{region '#Template'}
	{attribute 'Version' := '6.0.0.0'}
	{attribute 'Tags' := '"LCID": "1031", "Text": "RA, Sunprotection, Sunblind, Zone"'}
	{attribute 'Tags' := '"LCID": "1033", "Text": "RA, Sunprotection, Sunblind, Zone"'}
	{attribute 'Using' := '"Type": "Template", "URI": "ST_BA_Facade"'}
	{attribute 'Using' := '"Type": "Template", "URI": "ST_BA_SunblindActuatorFeedback"'}
	{attribute 'Description' := '"LCID": "1031", "Text": "Sonnenschutzlogik (Jalousie) für eine Zone (Raum)"'}
	{attribute 'Description' := '"LCID": "1033", "Text": "Sunblind-logic (venetian blind) for one zone (room)"'}
{endregion}
FUNCTION_BLOCK FB_BA_SunblindZone EXTENDS FB_BA_Ext_SunblindAngle
VAR_INPUT	
	fRoomTempSen			: REAL;
	bPrcDetc				: BOOL;
	bSwiUp					: BOOL;
	bSwiDwn					: BOOL;	      
	stBuildingSpRmT			: ST_BA_SpRmT;
	stFacade				: ST_BA_Facade;
	stScene					: ST_BA_Sunbld;
	stReferenceFeedback		: ST_BA_SunblindActuatorFeedback;
END_VAR                 
VAR_OUTPUT              
	stSunBldOut				: ST_BA_SunBld;			// command telegram
END_VAR
VAR_INPUT CONSTANT PERSISTENT
	bThAutoSlcn				: BOOL;		// Thermo-automatic enable
	{attribute 'parameterUnit':= '%'}       
	fThAutoColPos			: REAL;		// Thermo-automatic cooling-position [%]
	{attribute 'parameterUnit':= 'degree'}  
	fThAutoColAngl			: REAL;		// Thermo-automatic cooling-angle [deg]
		                                    
	bSunPrtcSlcn			: BOOL;		// Sun-Protection-automatic enable     
		                                    
	bTwiLgtAutoSlcn			: BOOL;		// Twilight-automatic enable
	{attribute 'parameterUnit':= '%'}        
	fTwiLgtAutoPos			: REAL;		// Twilight-automatic cooling-position [%]
	{attribute 'parameterUnit':= 'degree'}   
	fTwiLgtAutoAngl			: REAL;		// Twilight-automatic cooling-angle [deg]
	{attribute 'parameterUnit':= 's'}
	{attribute 'parameterUnit':= 'ms'}
	nSwiOverTi 				: UDINT;	// zone-manual-control: switch-over time from step to continous mode [ms]
END_VAR
VAR_INPUT CONSTANT
	ManSwi					: FB_BA_SunBldSwi:= (ePrio:= E_BA_SunBldPrio.eManualGroup);
	ThAuto					: FB_BA_SunBldEvt:= (ePrio:= E_BA_SunBldPrio.eGroupThermoAuto);	
	SunPrtc					: FB_BA_SunBldEvt:= (ePrio:= E_BA_SunBldPrio.eSunProtection);	
	TwiLgtAuto				: FB_BA_SunBldEvt:= (ePrio:= E_BA_SunBldPrio.eGroupTwiLightAuto);
END_VAR
VAR                       	                                                    
	ThAutoSwi				: FB_BA_Swi2P;                                    
	PrioSwi					: FB_BA_SunBldTgmSel8;
	EnSunBldSwi				: SR;
END_VAR
VAR // added by the converter: edge detectors and wires of the graphical bodies
    _w1 : BOOL;
END_VAR

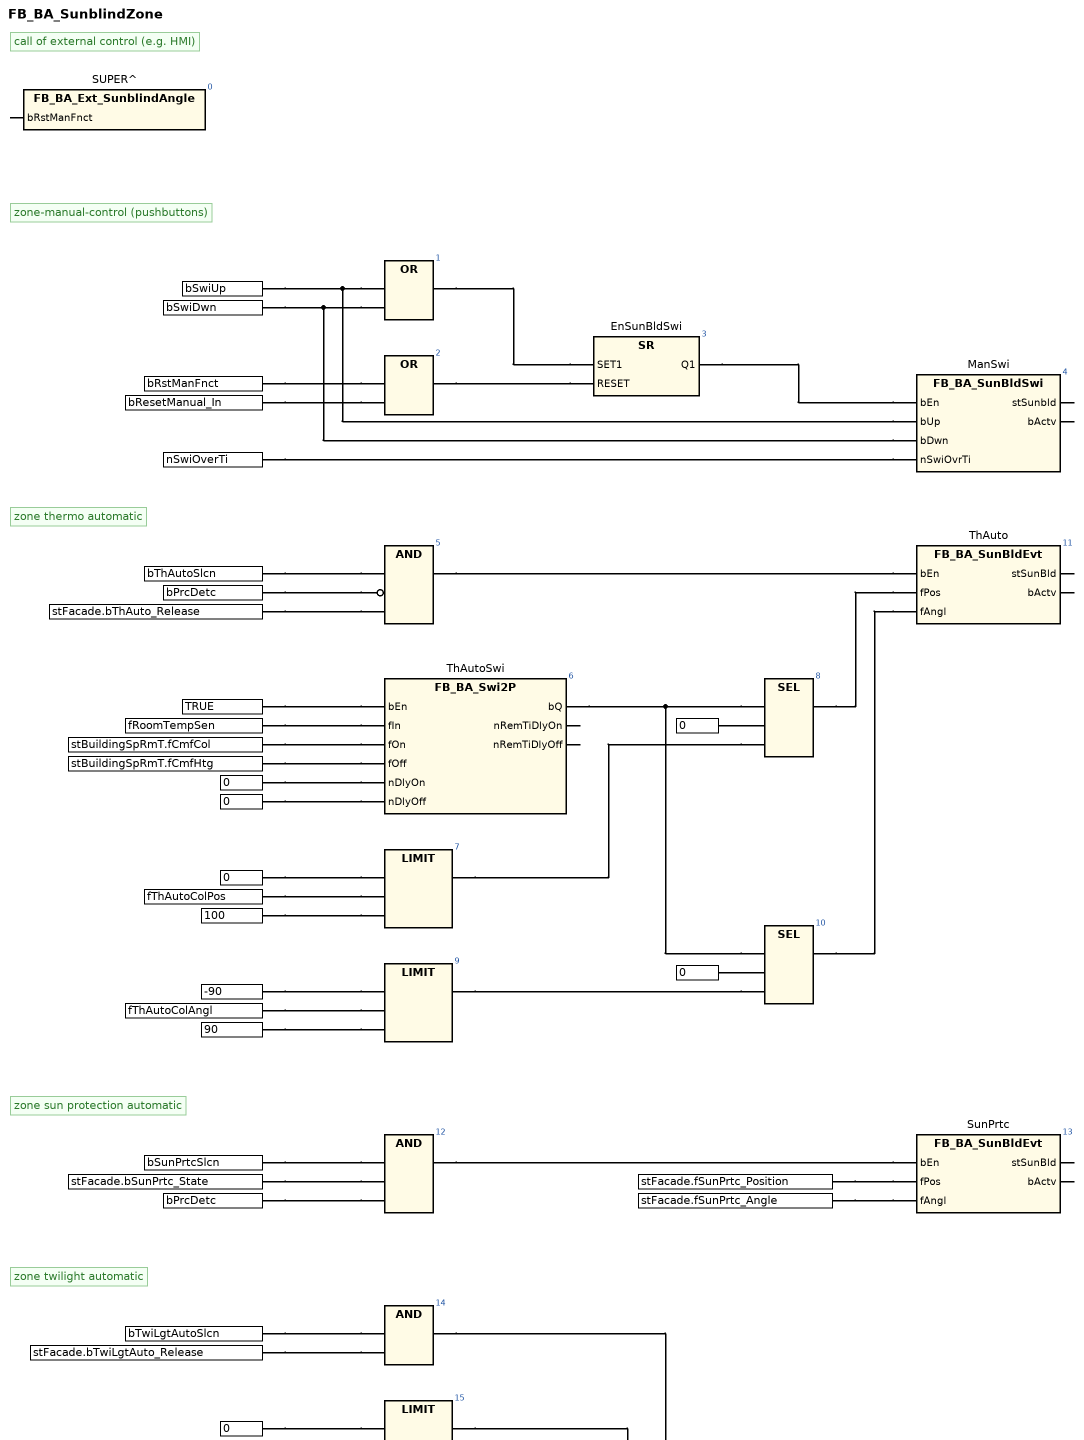
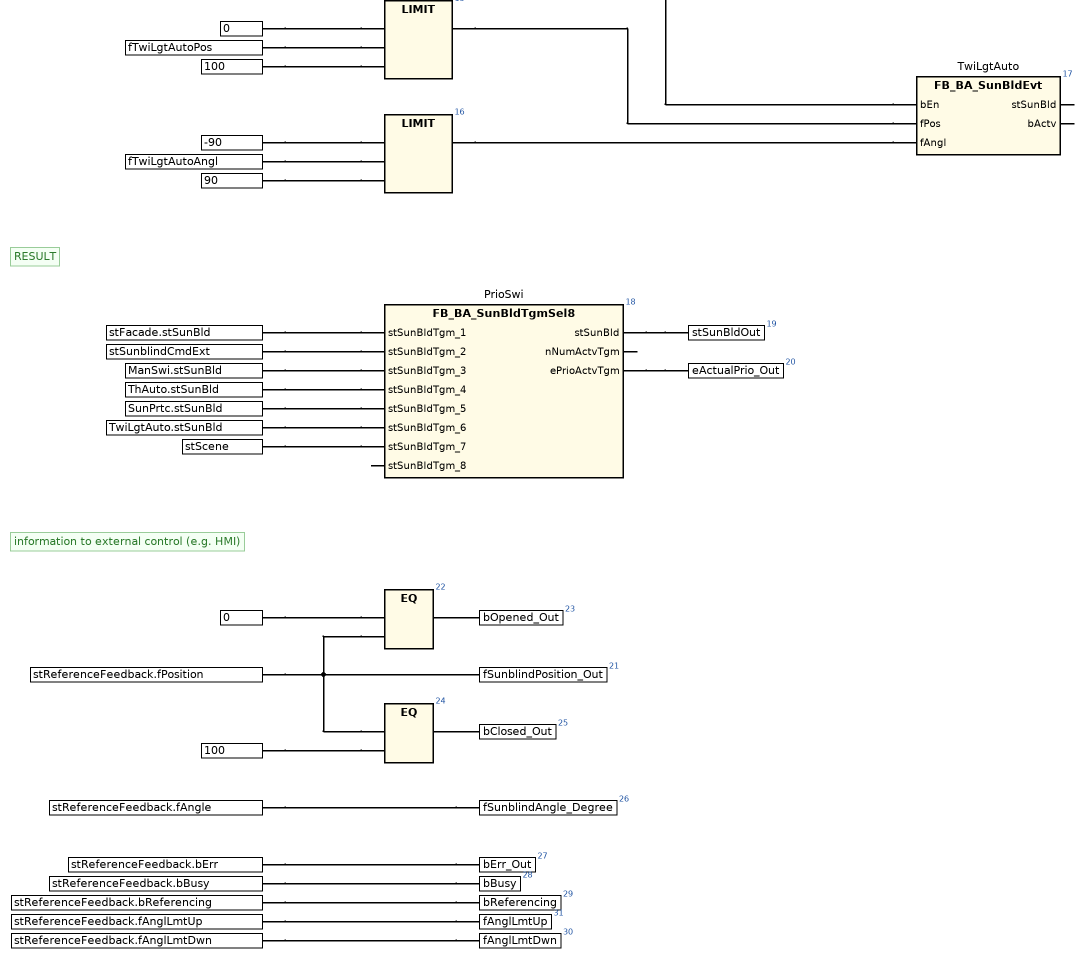
// call of external control (e.g. HMI)
SUPER^(); // FB_BA_Ext_SunblindAngle
// zone-manual-control (pushbuttons)
EnSunBldSwi(SET1 := bSwiUp OR bSwiDwn, RESET := bRstManFnct OR bResetManual_In); // SR
ManSwi(bEn := EnSunBldSwi.Q1, bUp := bSwiUp, bDwn := bSwiDwn, nSwiOvrTi := nSwiOverTi); // FB_BA_SunBldSwi
// zone thermo automatic
_w1 := bThAutoSlcn AND NOT bPrcDetc AND stFacade.bThAuto_Release;
ThAutoSwi(
    bEn := TRUE,
    fIn := fRoomTempSen,
    fOn := stBuildingSpRmT.fCmfCol,
    fOff := stBuildingSpRmT.fCmfHtg,
    nDlyOn := 0,
    nDlyOff := 0); // FB_BA_Swi2P
ThAuto(
    bEn := _w1,
    fPos := SEL(ThAutoSwi.bQ, 0, LIMIT(0, fThAutoColPos, 100)),
    fAngl := SEL(ThAutoSwi.bQ, 0, LIMIT(-90, fThAutoColAngl, 90))); // FB_BA_SunBldEvt
// zone sun protection automatic
SunPrtc(
    bEn := bSunPrtcSlcn AND stFacade.bSunPrtc_State AND bPrcDetc,
    fPos := stFacade.fSunPrtc_Position,
    fAngl := stFacade.fSunPrtc_Angle); // FB_BA_SunBldEvt
// zone twilight automatic
TwiLgtAuto(
    bEn := bTwiLgtAutoSlcn AND stFacade.bTwiLgtAuto_Release,
    fPos := LIMIT(0, fTwiLgtAutoPos, 100),
    fAngl := LIMIT(-90, fTwiLgtAutoAngl, 90)); // FB_BA_SunBldEvt
// RESULT
PrioSwi(
    stSunBldTgm_1 := stFacade.stSunBld,
    stSunBldTgm_2 := stSunblindCmdExt,
    stSunBldTgm_3 := ManSwi.stSunBld,
    stSunBldTgm_4 := ThAuto.stSunBld,
    stSunBldTgm_5 := SunPrtc.stSunBld,
    stSunBldTgm_6 := TwiLgtAuto.stSunBld,
    stSunBldTgm_7 := stScene); // FB_BA_SunBldTgmSel8
stSunBldOut := PrioSwi.stSunBld;
eActualPrio_Out := PrioSwi.ePrioActvTgm;
fSunblindPosition_Out := stReferenceFeedback.fPosition;
// information to external control (e.g. HMI)
bOpened_Out := 0 = stReferenceFeedback.fPosition;
bClosed_Out := stReferenceFeedback.fPosition = 100;
fSunblindAngle_Degree := stReferenceFeedback.fAngle;
bErr_Out := stReferenceFeedback.bErr;
bBusy := stReferenceFeedback.bBusy;
bReferencing := stReferenceFeedback.bReferencing;
fAnglLmtDwn := stReferenceFeedback.fAnglLmtDwn;
fAnglLmtUp := stReferenceFeedback.fAnglLmtUp;

METHOD FB_init : BOOL
VAR_INPUT
	bInitRetains : BOOL; // if TRUE; the retain variables are initialized (warm start / cold start)
	bInCopyCode : BOOL;  // if TRUE; the instance afterwards gets moved into the copy code (online change)
END_VAR
bThAutoSlcn				:= TRUE;							// Thermo-automatic enable
fThAutoColPos			:= 100.0;							// Thermo-automatic cooling-position [%]
fThAutoColAngl			:= -90.0;							// Thermo-automatic cooling-angle [deg]
bSunPrtcSlcn			:= TRUE;							// Sun-Protection-automatic enable     
bTwiLgtAutoSlcn			:= FALSE;							// Twilight-automatic enable
fTwiLgtAutoPos			:= 100.0;							// Twilight-automatic position [%]
fTwiLgtAutoAngl			:= -90.0;							// Twilight-automatic angle [deg]
nSwiOverTi 				:= 250;								// Zone-manual-control: switch-over time from step to continous mode [ms]
                        
ManSwi.ePrio			:= E_BA_SunBldPrio.eManualGroup;	// Priority of internal manual telegram
END_METHOD

END_FUNCTION_BLOCK

(* stored: Version 1.1.0.1, ProductVersion 3.1.4024.12
   POU FB_BA_SunblindZone: Id {e2d92f38-0fe4-41e3-8849-613ba5c7e027}, SpecialFunc None
   Method FB_init: Id {460e35d3-c44e-4476-8d37-6fdfbc7e6790} *)
